ABB RAPID module: Wobj_FRAME_PalletSaida.mod

MODULE Wobj_FRAME_PalletSaida
	! Points are read in order of declaration.
  ! Please do not change the order of points!

  LOCAL PERS robtarget pWobj_U_PointX1:=[[-2365.535,-1161.537,461.8855],[0.0839413478970528,-0.639336228370667,-0.705879032611847,0.293151468038559],[-2,0,-1,0],[9E+09,9E+09,9E+09,9E+09,9E+09,9E+09]];
	LOCAL PERS robtarget pWobj_U_PointX2:=[[-2377.297,-434.3304,464.501],[0.0839445516467094,-0.639337360858917,-0.705874800682068,0.293158292770386],[-2,0,-2,0],[9E+09,9E+09,9E+09,9E+09,9E+09,9E+09]];
	LOCAL PERS robtarget pWobj_U_PointY1:=[[-2993.311,-1168.85,465.0061],[0.0839396864175797,-0.639336228370667,-0.705880105495453,0.293149352073669],[-2,0,-1,0],[9E+09,9E+09,9E+09,9E+09,9E+09,9E+09]];

ENDMODULE
